// TIA Portal V21 export
// export: Created 2026-06-08T02:45:14.9987773Z, ExportSetting WithReadOnly, DisplayName Totally Integrated Automation Portal, DisplayVersion V21, DisplayName SINAMICS Startdrive Advanced, DisplayVersion V21, DisplayName SINAMICS Startdrive G110M, G120, G120C, G120D, G120P, G115D, DisplayVersion V21, DisplayName SINAMICS Startdrive G130, G150, S120, S150, G200, G220, S200, S210, S220, Innomotics MVD, DisplayVersion V21, DisplayName STEP 7 Professional, DisplayVersion V21, DisplayName STEP 7 Safety, DisplayVersion V21, DisplayName Tech WebApplication, DisplayVersion V21, DisplayName WinCC Basic/Comfort/Advanced, DisplayVersion V21, DisplayName WinCC Professional, DisplayVersion V21, DisplayName WinCC Unified, DisplayVersion V21
FUNCTION_BLOCK "FB_FertigationControl"   // FB2, SCL
{ S7_Optimized_Access := 'TRUE' }
// stored: CodeModifiedDate 2026-06-07T02:45:42.0628027Z, CompileDate 2026-06-07T02:45:42.0628027Z, CreationDate 2026-06-07T02:45:40.5967252Z, DownloadDate 2026-06-07T02:47:24.9117008Z, InterfaceModifiedDate 2026-06-07T02:45:40.6736502Z, IsConsistent true, LibraryConformanceStatus 该对象为库兼容。, LoadMemoryLength 26630, MemoryReserve 100, ModifiedDate 2026-06-07T02:45:42.0628027Z, PLCSimAdvancedSupport true, ParameterModified 2026-06-07T02:45:40.6736502Z, SetENOAutomatically false, StructureModified 2026-06-07T02:45:40.6736502Z, WorkMemoryLength 1166
   VAR_INPUT
      EC_Set_SP : Real;   // 上位机/SAC 目标 EC
      pH_Set_SP : Real;   // 上位机/SAC 目标 pH
      EC_Actual : Real;   // 出口 EC 反馈
      pH_Actual : Real;   // 出口 pH 反馈
      SAC_Enable : Bool;   // 远程控制使能
      Remote_Heartbeat : Int;   // 上位机心跳
      CycleTime : Real := 0.1;   // 调用周期，单位 s
      Kp_EC : Real := 4.0;   // EC PID 比例增益
      Ki_EC : Real := 0.25;   // EC PID 积分增益
      Kd_EC : Real := 0.0;   // EC PID 微分增益，联调初期先置 0
      Kp_pH : Real := 2.0;   // pH PID 比例增益，pH 偏高时加酸
      Ki_pH : Real := 0.15;   // pH PID 积分增益
      Kd_pH : Real := 0.0;   // pH PID 微分增益，联调初期先置 0
      EC_Filter_Tau : Real := 2.0;   // EC 反馈滤波时间常数，单位 s，越大越稳但响应越慢
      pH_Filter_Tau : Real := 3.0;   // pH 反馈滤波时间常数，单位 s
      q_f_min : Real := 0.0;
      q_f_max : Real := 10.0;
      q_a_min : Real := 0.0;
      q_a_max : Real := 4.0;
      Watchdog_Limit : Int := 10000;   // 心跳超限后进入安全输出，需大于两次 Python 写入间隔内的 OB1 扫描次数
   END_VAR
   VAR_OUTPUT
      Remote_Comms_OK : Bool;
      Watchdog_Timer : Int;
      q_f_cmd : Real;
      q_a_cmd : Real;
      Valve_F_Actual : Real;
      Valve_A_Actual : Real;
      AQ_Valve_F_Raw : Int;
      AQ_Valve_A_Raw : Int;
      System_Alarm_Light : Bool;
   END_VAR
   VAR
      Last_Heartbeat : Int;
      Watchdog_Count : Int;
      q_f_raw : Real;
      q_a_raw : Real;
      EC_Integral : Real;
      pH_Integral : Real;
      EC_Error_Last : Real;
      pH_Error_Last : Real;
      EC_Filtered : Real;
      pH_Filtered : Real;
      Filter_Init : Bool;
      inst_RL_F { S7_SetPoint := 'True'} : "RateLimiter";
      inst_RL_A { S7_SetPoint := 'True'} : "RateLimiter";
      tWatchdog : TON_TIME;
   END_VAR
   VAR_TEMP
      EC_Error : Real;
      pH_Error : Real;
      q_f_target : Real;
      q_a_target : Real;
      Heartbeat_Changed : Bool;
      EC_Derivative : Real;
      pH_Derivative : Real;
      q_f_pid : Real;
      q_a_pid : Real;
      EC_Alpha : Real;
      pH_Alpha : Real;
   END_VAR
BEGIN

      // ================================================================
      // B 方案 PLC 执行层
      // Python/SAC 只给 EC_set、pH_set；PLC 根据反馈计算 q_f、q_a。
      // 当前版本先用简单比例控制，跑通后可替换为 PID / ESO-AFOPID。
      // ================================================================

      // --- 心跳监控 ---
      // 参考旧 PLC 写法：不用 OB1 扫描次数判断通信，而用 TON 定时器判断。
      // Python 正常运行时 Remote_Heartbeat 会周期性变化，每次变化都复位 TON；
      // 超过 3 秒没有新心跳，才认为上位机通信中断。
      #Heartbeat_Changed := (#Remote_Heartbeat <> #Last_Heartbeat);

      IF #Heartbeat_Changed THEN
         #Last_Heartbeat := #Remote_Heartbeat;
         #Watchdog_Count := 0;
      ELSE
         #Watchdog_Count := #Watchdog_Count + 1;
      END_IF;

      #tWatchdog(IN := NOT #Heartbeat_Changed,
                 PT := T#3s);

      #Watchdog_Timer := #Watchdog_Count;
      #Remote_Comms_OK := NOT #tWatchdog.Q;

      // --- 安全状态：未使能或通讯超时，所有执行量归零 ---
      IF (NOT #SAC_Enable) OR (NOT #Remote_Comms_OK) THEN
         #q_f_raw := 0.0;
         #q_a_raw := 0.0;
         #q_f_cmd := 0.0;
         #q_a_cmd := 0.0;
         #Valve_F_Actual := 0.0;
         #Valve_A_Actual := 0.0;
         #AQ_Valve_F_Raw := 0;
         #AQ_Valve_A_Raw := 0;
         #System_Alarm_Light := NOT #Remote_Comms_OK;
         RETURN;
      END_IF;

      // --- 反馈滤波 ---
      // Python/传感器写入的 EC_Actual、pH_Actual 可能有瞬时抖动；
      // PID 使用滤波后的值，避免泵阀跟着噪声频繁调整。
      IF NOT #Filter_Init THEN
         #EC_Filtered := #EC_Actual;
         #pH_Filtered := #pH_Actual;
         #Filter_Init := TRUE;
      END_IF;

      IF (#CycleTime > 0.0) AND (#EC_Filter_Tau > 0.0) THEN
         #EC_Alpha := #CycleTime / (#EC_Filter_Tau + #CycleTime);
      ELSE
         #EC_Alpha := 1.0;
      END_IF;

      IF (#CycleTime > 0.0) AND (#pH_Filter_Tau > 0.0) THEN
         #pH_Alpha := #CycleTime / (#pH_Filter_Tau + #CycleTime);
      ELSE
         #pH_Alpha := 1.0;
      END_IF;

      // 基本量程保护：明显不合理的传感器值不进入滤波器。
      IF (#EC_Actual >= 0.0) AND (#EC_Actual <= 10.0) THEN
         #EC_Filtered := #EC_Filtered + #EC_Alpha * (#EC_Actual - #EC_Filtered);
      END_IF;

      IF (#pH_Actual >= 0.0) AND (#pH_Actual <= 14.0) THEN
         #pH_Filtered := #pH_Filtered + #pH_Alpha * (#pH_Actual - #pH_Filtered);
      END_IF;

      // --- PID 闭环控制 ---
      // EC 偏低：增加肥料母液流量；EC 偏高：减少肥料母液流量。
      #EC_Error := #EC_Set_SP - #EC_Filtered;

      // pH 偏高：增加酸液流量；pH 偏低：减少酸液流量。
      #pH_Error := #pH_Filtered - #pH_Set_SP;

      IF #CycleTime > 0.0 THEN
         #EC_Integral := #EC_Integral + #EC_Error * #CycleTime;
         #pH_Integral := #pH_Integral + #pH_Error * #CycleTime;

         #EC_Derivative := (#EC_Error - #EC_Error_Last) / #CycleTime;
         #pH_Derivative := (#pH_Error - #pH_Error_Last) / #CycleTime;
      ELSE
         #EC_Derivative := 0.0;
         #pH_Derivative := 0.0;
      END_IF;

      // 积分限幅，防止长时间饱和后积分过大。
      IF #EC_Integral > 5.0 THEN
         #EC_Integral := 5.0;
      ELSIF #EC_Integral < -5.0 THEN
         #EC_Integral := -5.0;
      END_IF;

      IF #pH_Integral > 5.0 THEN
         #pH_Integral := 5.0;
      ELSIF #pH_Integral < -5.0 THEN
         #pH_Integral := -5.0;
      END_IF;

      // PID 增量叠加到上一周期执行量。
      #q_f_pid := #Kp_EC * #EC_Error + #Ki_EC * #EC_Integral + #Kd_EC * #EC_Derivative;
      #q_a_pid := #Kp_pH * #pH_Error + #Ki_pH * #pH_Integral + #Kd_pH * #pH_Derivative;

      #q_f_target := #q_f_raw + #q_f_pid;
      #q_a_target := #q_a_raw + #q_a_pid;

      #EC_Error_Last := #EC_Error;
      #pH_Error_Last := #pH_Error;

      // --- 物理限幅 ---
      IF #q_f_target < #q_f_min THEN
         #q_f_target := #q_f_min;
      ELSIF #q_f_target > #q_f_max THEN
         #q_f_target := #q_f_max;
      END_IF;

      IF #q_a_target < #q_a_min THEN
         #q_a_target := #q_a_min;
      ELSIF #q_a_target > #q_a_max THEN
         #q_a_target := #q_a_max;
      END_IF;

      // --- 斜坡限速，保护泵阀 ---
      #inst_RL_F(
         target := #q_f_target,
         maxRateUp := 2.0,
         maxRateDown := 3.0,
         cycleTime := #CycleTime,
         enable := TRUE,
         reset := FALSE
      );

      #inst_RL_A(
         target := #q_a_target,
         maxRateUp := 1.0,
         maxRateDown := 2.0,
         cycleTime := #CycleTime,
         enable := TRUE,
         reset := FALSE
      );

      #q_f_cmd := #inst_RL_F.output;
      #q_a_cmd := #inst_RL_A.output;
      #q_f_raw := #q_f_cmd;
      #q_a_raw := #q_a_cmd;

      #Valve_F_Actual := #q_f_cmd;
      #Valve_A_Actual := #q_a_cmd;

      // --- 0~27648 模拟量换算 ---
      #AQ_Valve_F_Raw := REAL_TO_INT(#q_f_cmd / #q_f_max * 27648.0);
      #AQ_Valve_A_Raw := REAL_TO_INT(#q_a_cmd / #q_a_max * 27648.0);

      #System_Alarm_Light := FALSE;
END_FUNCTION_BLOCK
